// TwinCAT 3 PLC project Main
// ProgramVersion: 3.1.4024.0
// libraries:
//   Tc2_Standard, * (Beckhoff Automation GmbH)
//   Tc2_System, * (Beckhoff Automation GmbH)
//   Tc2_Utilities, * (Beckhoff Automation GmbH)
//   Tc3_Module, * (Beckhoff Automation GmbH)
//   TcUnit, * (www.tcunit.org)
//   mobject-core,0.5.0,mobject
//   mobject-graph-plc-pack,0.15.0,mobject
// project tree:
//   / PlcTask.TcTTO (not stored)
//   POUs/ MAIN.TcPOU
//   Tests/Alias/ _FLOAT_TestSuite.TcPOU (not stored), _HRESULT_TestSuite.TcPOU
//   Tests/Arrays/ _Array0to7OfByte_TestSuite.TcPOU
//   Tests/Enums/ _E_TcEventClass_TestSuite.TcPOU
//   Tests/Structs/ _GUID_TestSuite.TcPOU, _TIMESTRUCT_TestSuite.TcPOU
// real-time tasks:
//   TASK PlcTask: cycle T#10ms, priority 20, ADS port 350

// ---- POUs/MAIN.TcPOU
PROGRAM MAIN
VAR
	
	//alias
    _FLOAT_TestSuite : _FLOAT_TestSuite;
	_HRESULT_TestSuite : _HRESULT_TestSuite;
	
	// arrays
	_Array0to7OfByte_TestSuite : _Array0to7OfByte_TestSuite;
    
	// struct
	_TIMESTRUCT_TestSuite : _TIMESTRUCT_TestSuite;
	_GUID_TestSuite : _GUID_TestSuite;
	
	// enums
	_E_TcEventClass_TestSuite : _E_TcEventClass_TestSuite;
	
END_VAR

TcUnit.RUN();

END_PROGRAM

// ---- Tests/Alias/_HRESULT_TestSuite.TcPOU
FUNCTION_BLOCK _HRESULT_TestSuite EXTENDS TcUnit.FB_TestSuite
VAR
END_VAR

TestAddress();
TestClearReference();
TestClone();
TestTypeNameReturnsExpected();
TestIdentifierReturnsExpected();
TestMakeReferenceToFollowsReference();
TestMakeReferenceToUpdatesReference();
TestSize();
TestValueReturnsExpectedAfterInit();
TestValueReturnsExpectedAfterChange();
TestSerializeTypeWith();
TestSerializeWith();
TestTryDeserializeFrom();
TestTryMakeReferenceToFollowsReference();
TestTryMakeReferenceToUpdatesReference();

METHOD PUBLIC TestAddress
VAR
    _type : _HRESULT(S_OK);
    notExpected : PVOID := 0;
    actual : PVOID;
END_VAR
TEST('TestAddress');

actual := _type.Address;

AssertFalse(
    Condition := (notExpected = actual),
    Message := 'Type did not return a valid address.'
);

TEST_FINISHED();
END_METHOD

METHOD PUBLIC TestClearReference
VAR
    _type : _HRESULT(S_OK);
	target : HRESULT := S_OK;
    expected : HRESULT := S_OK;
    actual : HRESULT;
END_VAR
TEST('TestClearReference');

_type.MakeReferenceTo(target);
_type.ClearReference();
target := S_FALSE;

actual := _type.Value;

AssertEquals(
    Expected := expected,
    Actual := actual,
    Message := 'Value did not follow target change'
);

TEST_FINISHED();
END_METHOD

METHOD PUBLIC TestClone
VAR
    _type : _HRESULT(S_OK);
	clone : I_Datatype;
	isValidClone : BOOL;
	compareResult : DINT;
END_VAR
TEST('TestClone');

clone := _type.Clone();

isValidClone := clone <> 0;

IF isValidClone THEN
	compareResult := memcmp(_type.Address, clone.Address, clone.Size);
END_IF

AssertTrue(
	Condition := isValidClone,
	Message := 'Clone did not produce a clone'
);

AssertEquals_DINT(
	Expected := 0,
    Actual := compareResult,
    Message := 'Clone did not return a valid clone.'
);

clone.Dispose();

TEST_FINISHED();
END_METHOD

METHOD PUBLIC TestIdentifierReturnsExpected
VAR
    _type : _HRESULT(S_OK);
    expected : STRING := 'HRESULT';
    actual : STRING;
END_VAR
TEST('TestIdentifierReturnsExpected');

actual := _type.Identifier;

AssertEquals_STRING(
    Expected := expected,
    Actual := actual,
    Message := 'Type did not return correct iec type.'
);

TEST_FINISHED();
END_METHOD

METHOD PUBLIC TestMakeReferenceToFollowsReference
VAR
    _type : _HRESULT(S_OK);
	target : HRESULT := S_OK;
    expected : HRESULT := S_FALSE;
    actual : HRESULT;
END_VAR
TEST('TestMakeReferenceToFollowsReference');

_type.MakeReferenceTo(target);
target := S_FALSE;

actual := _type.Value;

AssertEquals(
    Expected := expected,
    Actual := actual,
    Message := 'Value did not follow target change'
);

TEST_FINISHED();
END_METHOD

METHOD PUBLIC TestMakeReferenceToUpdatesReference
VAR
    _type : _HRESULT(S_OK);
	target : HRESULT := S_OK;
    expected : HRESULT := S_FALSE;
    actual : HRESULT;
END_VAR
TEST('TestMakeReferenceToUpdatesReference');

_type.MakeReferenceTo(target);
_type.Value := S_FALSE;

actual := target;

AssertEquals(
    Expected := expected,
    Actual := actual,
    Message := 'Value did not update target'
);

TEST_FINISHED();
END_METHOD

METHOD PUBLIC TestSerializeTypeWith
VAR
    _type : _HRESULT(S_OK);
    serializer : JsonSerializer;
    expected : STRING(500) := '{"typeName":"ALIAS","identifier":"HRESULT","baseDatatype":{"typeName":"DINT","minValue":-2147483648,"maxValue":2147483647,"isSigned":true,"isFloat":false}}';
    actual : STRING(500);
END_VAR
TEST('TestSerializeTypeWith');

serializer.Reset();
_type.SerializeTypeWith(serializer);
serializer.TryGetSerializedData(ADR(actual), SIZEOF(actual));

AssertEquals_STRING(
    Expected := expected,
    Actual := actual,
    Message := 'Serialization of type did not return correct string.'
);

TEST_FINISHED();
END_METHOD

METHOD PUBLIC TestSerializeWith
VAR
    _type : _HRESULT(S_FALSE);
    serializer : JsonSerializer;
    expected : STRING := '1';
    actual : STRING(500);
END_VAR
TEST('TestSerializeWith');

serializer.Reset();
_type.SerializeWith(serializer);
serializer.TryGetSerializedData(ADR(actual), SIZEOF(actual));

AssertEquals_STRING(
    Expected := expected,
    Actual := actual,
    Message := 'Serialization of type data did not return correct string.'
);

TEST_FINISHED();
END_METHOD

METHOD PUBLIC TestSize
VAR
    _type : _HRESULT(S_OK);
    expected : UDINT := SIZEOF(HRESULT);
    actual : UDINT;
END_VAR
TEST('TestSize');

actual := _type.Size;

AssertEquals_UDINT(
    Expected := Expected,
    Actual := actual,
    Message := 'Type did not return the correct size.'
);

TEST_FINISHED();
END_METHOD

METHOD PUBLIC TestTryDeserializeFrom
VAR
    deserializer : JsonDeserializer;
    feedback : DeserializerFeedback;
    json : STRING := '0';
    _type : _HRESULT(S_OK);
    expected : HRESULT := S_OK;
    actual : HRESULT;
 END_VAR
TEST('TestTryDeserializeFrom');

deserializer.Reset();
deserializer.TryLoad(json);
_type.TryDeserializeFrom(Deserializer, Feedback);

actual := _type.Value;

AssertEquals(
    Expected := expected,
    Actual := actual,
    Message := 'Type did not deserialize correctly.'
);

TEST_FINISHED();
END_METHOD

METHOD PUBLIC TestTryMakeReferenceToFollowsReference
VAR
    _type : _HRESULT(S_OK);
	target : _HRESULT(S_OK);
    expected : HRESULT := S_FALSE;
    actual : HRESULT;
END_VAR
TEST('TestTryMakeReferenceToFollowsReference');

_type.TryMakeReferenceTo(target);
target.Value := S_FALSE;

actual := _type.Value;

AssertEquals(
    Expected := expected,
    Actual := actual,
    Message := 'Value did not follow target change'
);

TEST_FINISHED();
END_METHOD

METHOD PUBLIC TestTryMakeReferenceToUpdatesReference
VAR
    _type : _HRESULT(S_OK);
	target : _HRESULT(S_OK);
    expected : HRESULT := S_FALSE;
    actual : HRESULT;
END_VAR
TEST('TestTryMakeReferenceToUpdatesReference');

_type.TryMakeReferenceTo(target);
_type.Value := S_FALSE;

actual := target.Value;

AssertEquals(
    Expected := expected,
    Actual := actual,
    Message := 'Value did not update target'
);

TEST_FINISHED();
END_METHOD

METHOD PUBLIC TestTypeNameReturnsExpected
VAR
    _type : _HRESULT(S_OK);
    expected : STRING := 'ALIAS';
    actual : STRING;
END_VAR
TEST('TestTypeNameReturnsExpected');

actual := _type.TypeName;

AssertEquals_STRING(
    Expected := expected,
    Actual := actual,
    Message := 'Type did not return correct iec type.'
);

TEST_FINISHED();
END_METHOD

METHOD PUBLIC TestValueReturnsExpectedAfterChange
VAR
    _type : _HRESULT(S_OK);
    expected : HRESULT := S_FALSE;
    actual : HRESULT;
END_VAR
TEST('TestValueReturnsExpectedAfterChange');

_type.Value := S_FALSE;

actual := _type.Value;

AssertEquals(
    Expected := expected,
    Actual := actual,
    Message := 'Expected value not returned after change.'
);

TEST_FINISHED();
END_METHOD

METHOD PUBLIC TestValueReturnsExpectedAfterInit
VAR
    _type : _HRESULT(S_FALSE);
    expected : HRESULT := S_FALSE;
    actual : HRESULT;
END_VAR
TEST('TestValueReturnsExpectedAfterInit');

actual := _type.Value;

AssertEquals(
    Expected := expected,
    Actual := actual,
    Message := 'Expected value not returned after Init.'
);

TEST_FINISHED();
END_METHOD

END_FUNCTION_BLOCK

// ---- Tests/Arrays/_Array0to7OfByte_TestSuite.TcPOU
FUNCTION_BLOCK _Array0to7OfByte_TestSuite EXTENDS TcUnit.FB_TestSuite
VAR
END_VAR

TestAddress();
TestBaseDatatype();
TestClearReference();
TestClone();
TestTypeNameReturnsExpected();
TestIdentifierReturnsExpected();
TestLength();
TestLowerBound();
TestLowerBoundWithInvalidDimention();
TestMakeReferenceToFollowsReference();
TestMakeReferenceToUpdatesReference();
TestSize();
TestSerializeTypeWith();
TestSerializeWith();
TestTryDeserializeFrom();
TestTryGetElementAsDatatypeWithInvalidDimentionTooBig();
TestTryGetElementAsDatatypeWithInvalidDimentionTooSmall();
TestTryMakeReferenceToFollowsReference();
TestTryMakeReferenceToUpdatesReference();
TestUpperBound();
TestUpperBoundWithInvalidDimention();
TestValueReturnsExpectedAfterChange();

METHOD PUBLIC TestAddress
VAR
    _type : _Array0to7OfByte;
    notExpected : PVOID := 0;
    actual : PVOID;
END_VAR
TEST('TestAddress');

actual := _type.Address;

AssertFalse(
    Condition := (notExpected = actual),
    Message := 'Type did not return a valid address.'
);

TEST_FINISHED();
END_METHOD

METHOD PUBLIC TestBaseDatatype
VAR
    _type : _Array0to7OfByte;
    expected : T_MAXSTRING := 'BYTE';
    actual : T_MAXSTRING;
END_VAR
TEST('TestBaseDatatype');

actual := _type.BaseDatatype.TypeName;

AssertEquals_STRING(
    Expected := expected,
    Actual := actual,
    Message := 'Type did not return the correct base type'
);

TEST_FINISHED();
END_METHOD

METHOD PUBLIC TestClearReference
VAR
    _type : _Array0to7OfByte;
	target : ARRAY [0..7] OF BYTE;
    expected : ARRAY [0..7] OF BYTE := [0,0,0,0,0,0,0,0];
    actual : ARRAY [0..7] OF BYTE;
END_VAR
TEST('TestClearReference');

_type.MakeReferenceTo(target);
_type.ClearReference();
target[5] := 123;

actual := _type.Value;

AssertEquals(
    Expected := expected,
    Actual := actual,
    Message := 'Value incorrectly followed target change'
);

TEST_FINISHED();
END_METHOD

METHOD PUBLIC TestClone
VAR
    _type : _Array0to7OfByte;
	clone : I_Datatype;
	isValidClone : BOOL;
	compareResult : DINT;
END_VAR
TEST('TestClone');

clone := _type.Clone();

isValidClone := clone <> 0;

IF isValidClone THEN
	compareResult := memcmp(_type.Address, clone.Address, clone.Size);
END_IF

AssertTrue(
	Condition := isValidClone,
	Message := 'Clone did not produce a clone'
);

AssertEquals_DINT(
	Expected := 0,
    Actual := compareResult,
    Message := 'Clone did not return a valid clone.'
);

clone.Dispose();

TEST_FINISHED();
END_METHOD

METHOD PUBLIC TestIdentifierReturnsExpected
VAR
    _type : _Array0to7OfByte;
    expected : STRING := 'ARRAY [0..7] OF BYTE';
    actual : STRING;
END_VAR
TEST('TestIdentifierReturnsExpected');

actual := _type.Identifier;

AssertEquals_STRING(
    Expected := expected,
    Actual := actual,
    Message := 'Type did not return correct iec type.'
);

TEST_FINISHED();
END_METHOD

METHOD PUBLIC TestLength
VAR
    _type : _Array0to7OfByte;
    expected : UDINT := 8;
    actual : UDINT;
END_VAR
TEST('TestLength');

actual := _type.Length;

AssertEquals_UDINT(
    Expected := Expected,
    Actual := actual,
    Message := 'Type did not return the correct array length.'
);

TEST_FINISHED();
END_METHOD

METHOD PUBLIC TestLowerBound
VAR
    _type : _Array0to7OfByte;
    expected : DINT := 0;
    actual : DINT;
	ok : BOOL;
END_VAR
TEST('TestLowerBound');

ok := _type.TryGetLowerBound(1, actual);

AssertTrue(
    Condition := ok,
    Message := 'Type did not indicate that lower bound was possible to retreive.'
);

AssertEquals_DINT(
    Expected := Expected,
    Actual := actual,
    Message := 'Type did not return the correct array lower bound.'
);

TEST_FINISHED();
END_METHOD

METHOD PUBLIC TestLowerBoundWithInvalidDimention
VAR
    _type : _Array0to7OfByte;
    actual : DINT;
	result : BOOL;
END_VAR
TEST('TestLowerBoundWithInvalidDimention');

result := _type.TryGetLowerBound(2, actual);

AssertFalse(
    Condition := result,
    Message := 'Type did not indicate that the dimention was invalid'
);

TEST_FINISHED();
END_METHOD

METHOD PUBLIC TestMakeReferenceToFollowsReference
VAR
	_type : _Array0to7OfByte;
	target : ARRAY [0..7] OF BYTE;
    expected : ARRAY [0..7] OF BYTE := [1,2,3,4,5,6,7,8];
    actual : ARRAY [0..7] OF BYTE;
END_VAR
TEST('TestMakeReferenceToFollowsReference');

_type.MakeReferenceTo(target);
target[0] := 1;
target[1] := 2;
target[2] := 3;
target[3] := 4;
target[4] := 5;
target[5] := 6;
target[6] := 7;
target[7] := 8;

actual := _type.Value;

AssertEquals(
    Expected := expected,
    Actual := actual,
    Message := 'Value did not follow target change'
);

TEST_FINISHED();
END_METHOD

METHOD PUBLIC TestMakeReferenceToUpdatesReference
VAR
	_type : _Array0to7OfByte;
	target : ARRAY [0..7] OF BYTE;
    expected : ARRAY [0..7] OF BYTE := [1,2,3,4,5,6,7,8];
    actual : ARRAY [0..7] OF BYTE;
END_VAR
TEST('TestMakeReferenceToUpdatesReference');

_type.MakeReferenceTo(target);
target[0] := 1;
target[1] := 2;
target[2] := 3;
target[3] := 4;
target[4] := 5;
target[5] := 6;
target[6] := 7;
target[7] := 8;

actual := target;

AssertEquals(
    Expected := expected,
    Actual := actual,
    Message := 'Value did not update target'
);

TEST_FINISHED();
END_METHOD

METHOD PUBLIC TestSerializeTypeWith
VAR
    _type : _Array0to7OfByte;
    serializer : JsonSerializer;
    expected : STRING(1000) := '{"typeName":"ARRAY","identifier":"ARRAY [0..7] OF BYTE","baseType":{"typeName":"BYTE","minValue":0,"maxValue":255,"isSigned":false,"isFloat":false}}';
    actual : STRING(1000);
END_VAR
TEST('TestSerializeTypeWith');

serializer.Reset();
_type.SerializeTypeWith(serializer);
serializer.TryGetSerializedData(ADR(actual), SIZEOF(actual));

AssertEquals_STRING(
    Expected := expected,
    Actual := actual,
    Message := 'Serialization of type did not return correct string.'
);

TEST_FINISHED();
END_METHOD

METHOD PUBLIC TestSerializeWith
VAR
    _type : _Array0to7OfByte;
    serializer : JsonSerializer;
    expected : STRING(500) := '[1,2,3,4,5,6,7,8]';
    actual : STRING(500);
END_VAR
TEST('TestSerializeWith');

_type.Value[0] := 1;
_type.Value[1] := 2;
_type.Value[2] := 3;
_type.Value[3] := 4;
_type.Value[4] := 5;
_type.Value[5] := 6;
_type.Value[6] := 7;
_type.Value[7] := 8;

serializer.Reset();
_type.SerializeWith(serializer);
serializer.TryGetSerializedData(ADR(actual), SIZEOF(actual));

AssertEquals_STRING(
    Expected := expected,
    Actual := actual,
    Message := 'Serialization of type data did not return correct string.'
);

TEST_FINISHED();
END_METHOD

METHOD PUBLIC TestSize
VAR
    _type : _Array0to7OfByte;
	example : ARRAY [0..7] OF BYTE;
    expected : UDINT := SIZEOF(example);
    actual : UDINT;
END_VAR
TEST('TestSize');

actual := _type.Size;

AssertEquals_UDINT(
    Expected := Expected,
    Actual := actual,
    Message := 'Type did not return the correct size.'
);

TEST_FINISHED();
END_METHOD

METHOD PUBLIC TestTryDeserializeFrom
VAR
    deserializer : JsonDeserializer;
    feedback : DeserializerFeedback;
    json : STRING(500) := '[1,2,3,4,5,6,7,8]';
    _type : _Array0to7OfByte;
    expected :  ARRAY [0..7] OF BYTE := [1,2,3,4,5,6,7,8];
    actual : ARRAY [0..7] OF BYTE;
 END_VAR
TEST('TestTryDeserializeFrom');

deserializer.Reset();
deserializer.TryLoad(json);
_type.TryDeserializeFrom(Deserializer, Feedback);

actual := _type.Value;

AssertEquals(
    Expected := expected,
    Actual := actual,
    Message := 'Type did not deserialize correctly.'
);

TEST_FINISHED();
END_METHOD

METHOD PUBLIC TestTryGetElementAsDatatypeWithInvalidDimentionTooBig
VAR
    _type : _Array0to7OfByte;
    actual : I_Datatype;
	result : BOOL;
END_VAR
TEST('TestTryGetElementAsDatatypeWithInvalidDimentionTooBig');

result := _type.TryGetElementAsDatatypeByIndex(11, actual);

AssertFalse(
    Condition := result,
    Message := 'Type did not indicate that the dimention was invalid'
);

TEST_FINISHED();
END_METHOD

METHOD PUBLIC TestTryGetElementAsDatatypeWithInvalidDimentionTooSmall
VAR
    _type : _Array0to7OfByte;
    actual : I_Datatype;
	result : BOOL;
END_VAR
TEST('TestTryGetElementAsDatatypeWithInvalidDimentionTooSmall');

result := _type.TryGetElementAsDatatypeByIndex(-1, actual);

AssertFalse(
    Condition := result,
    Message := 'Type did not indicate that the dimention was invalid'
);

TEST_FINISHED();
END_METHOD

METHOD PUBLIC TestTryMakeReferenceToFollowsReference
VAR
    _type : _Array0to7OfByte;
	target : _Array0to7OfByte;
    expected : ARRAY [0..7] OF BYTE := [1,2,3,4,5,6,7,8];
    actual :  ARRAY [0..7] OF BYTE;
END_VAR
TEST('TestTryMakeReferenceToFollowsReference');

_type.TryMakeReferenceTo(target);
target.Value[0] := 1;
target.Value[1] := 2;
target.Value[2] := 3;
target.Value[3] := 4;
target.Value[4] := 5;
target.Value[5] := 6;
target.Value[6] := 7;
target.Value[7] := 8;

actual := _type.Value;

AssertEquals(
    Expected := expected,
    Actual := actual,
    Message := 'Value did not follow target change'
);

TEST_FINISHED();
END_METHOD

METHOD PUBLIC TestTryMakeReferenceToUpdatesReference
VAR
    _type : _Array0to7OfByte;
	target : _Array0to7OfByte;
    expected : ARRAY [0..7] OF BYTE := [1,2,3,4,5,6,7,8];
    actual :  ARRAY [0..7] OF BYTE;
END_VAR
TEST('TestTryMakeReferenceToUpdatesReference');

_type.TryMakeReferenceTo(target);
_type.Value[0] := 1;
_type.Value[1] := 2;
_type.Value[2] := 3;
_type.Value[3] := 4;
_type.Value[4] := 5;
_type.Value[5] := 6;
_type.Value[6] := 7;
_type.Value[7] := 8;

actual := target.Value;

AssertEquals(
    Expected := expected,
    Actual := actual,
    Message := 'Value did not update target'
);

TEST_FINISHED();
END_METHOD

METHOD PUBLIC TestTypeNameReturnsExpected
VAR
    _type : _Array0to7OfByte;
    expected : STRING := 'ARRAY';
    actual : STRING;
END_VAR
TEST('TestTypeNameReturnsExpected');

actual := _type.TypeName;

AssertEquals_STRING(
    Expected := expected,
    Actual := actual,
    Message := 'Type did not return correct iec type.'
);

TEST_FINISHED();
END_METHOD

METHOD PUBLIC TestUpperBound
VAR
    _type : _Array0to7OfByte;
    expected : DINT := 7;
    actual : DINT;
	ok : BOOL;
END_VAR
TEST('TestUpperBound');

ok := _type.TryGetUpperBound(1, actual);

AssertTrue(
    Condition := ok,
    Message := 'Type did not indicate that upper bound was possible to retreive.'
);

AssertEquals_DINT(
    Expected := Expected,
    Actual := actual,
    Message := 'Type did not return the correct array upper bound.'
);

TEST_FINISHED();
END_METHOD

METHOD PUBLIC TestUpperBoundWithInvalidDimention
VAR
    _type : _Array0to7OfByte;
    actual : DINT;
	result : BOOL;
END_VAR
TEST('TestUpperBoundWithInvalidDimention');

result := _type.TryGetUpperBound(2, actual);

AssertFalse(
    Condition := result,
    Message := 'Type did not indicate that the dimention was invalid'
);

TEST_FINISHED();
END_METHOD

METHOD PUBLIC TestValueReturnsExpectedAfterChange
VAR
    _type : _Array0to7OfByte;
	value : ARRAY [0..7] OF BYTE := [1,2,3,4,5,6,7,8];
    expected : ARRAY [0..7] OF BYTE := [1,2,3,4,5,6,7,8];
    actual :  ARRAY [0..7] OF BYTE;
END_VAR
TEST('TestValueReturnsExpectedAfterChange');

_type.Value := value;
actual := _type.Value;

AssertEquals(
    Expected := expected,
    Actual := actual,
    Message := 'Expected value not returned after change.'
);

TEST_FINISHED();
END_METHOD

END_FUNCTION_BLOCK

// ---- Tests/Structs/_TIMESTRUCT_TestSuite.TcPOU
FUNCTION_BLOCK _TIMESTRUCT_TestSuite EXTENDS TcUnit.FB_TestSuite
VAR
END_VAR

TestAddress();
TestClearReference();
TestClone();
TestTypeNameReturnsExpected();
TestIdentifierReturnsExpected();
TestMakeReferenceToFollowsReference();
TestMakeReferenceToUpdatesReference();
TestSize();
TestValueReturnsExpectedAfterChange();
TestSerializeTypeWith();
TestSerializeWith();
TestTryDeserializeFrom();
TestTryMakeReferenceToFollowsReference();
TestTryMakeReferenceToUpdatesReference();

METHOD PUBLIC TestAddress
VAR
    _type : _TIMESTRUCT;
    notExpected : PVOID := 0;
    actual : PVOID;
END_VAR
TEST('TestAddress');

actual := _type.Address;

AssertFalse(
    Condition := (notExpected = actual),
    Message := 'Type did not return a valid address.'
);

TEST_FINISHED();
END_METHOD

METHOD PUBLIC TestClearReference
VAR
    _type : _TIMESTRUCT;
	target : TIMESTRUCT;
    expected : TIMESTRUCT;
    actual : TIMESTRUCT;
END_VAR
TEST('TestClearReference');

_type.MakeReferenceTo(target);
_type.ClearReference();
target.wDay := 2;

actual := _type.Value;

AssertEquals(
    Expected := expected,
    Actual := actual,
    Message := 'Value did not follow target change'
);

TEST_FINISHED();
END_METHOD

METHOD PUBLIC TestClone
VAR
    _type : _TIMESTRUCT;
	clone : I_Datatype;
	isValidClone : BOOL;
	compareResult : DINT;
END_VAR
TEST('TestClone');

clone := _type.Clone();

isValidClone := clone <> 0;

IF isValidClone THEN
	compareResult := memcmp(_type.Address, clone.Address, clone.Size);
END_IF

AssertTrue(
	Condition := isValidClone,
	Message := 'Clone did not produce a clone'
);

AssertEquals_DINT(
	Expected := 0,
    Actual := compareResult,
    Message := 'Clone did not return a valid clone.'
);

clone.Dispose();

TEST_FINISHED();
END_METHOD

METHOD PUBLIC TestIdentifierReturnsExpected
VAR
    _type : _TIMESTRUCT;
    expected : STRING := 'TIMESTRUCT';
    actual : STRING;
END_VAR
TEST('TestIdentifierReturnsExpected');

actual := _type.Identifier;

AssertEquals_STRING(
    Expected := expected,
    Actual := actual,
    Message := 'Type did not return correct iec type.'
);

TEST_FINISHED();
END_METHOD

METHOD PUBLIC TestMakeReferenceToFollowsReference
VAR
    _type : _TIMESTRUCT;
	target : TIMESTRUCT;
    expected : TIMESTRUCT := (wDay := 2);
    actual : TIMESTRUCT;
END_VAR
TEST('TestMakeReferenceToFollowsReference');

_type.MakeReferenceTo(target);
target.wDay := 2;

actual := _type.Value;

AssertEquals(
    Expected := expected,
    Actual := actual,
    Message := 'Value did not follow target change'
);

TEST_FINISHED();
END_METHOD

METHOD PUBLIC TestMakeReferenceToUpdatesReference
VAR
    _type : _TIMESTRUCT;
	target : TIMESTRUCT;
    expected : TIMESTRUCT := (wDay := 2);
    actual : TIMESTRUCT;
END_VAR
TEST('TestMakeReferenceToUpdatesReference');

_type.MakeReferenceTo(target);
_type.wDay.Value := 2;

actual := target;

AssertEquals(
    Expected := expected,
    Actual := actual,
    Message := 'Value did not update target'
);

TEST_FINISHED();
END_METHOD

METHOD PUBLIC TestSerializeTypeWith
VAR
    _type : _TIMESTRUCT;
    serializer : JsonSerializer;
    expected : STRING(1000) := '{"typeName":"STRUCT","identifier":"TIMESTRUCT","members":{"wYear":{"typeName":"WORD","minValue":0,"maxValue":65535,"isSigned":false,"isFloat":false},"wMonth":{"typeName":"WORD","minValue":0,"maxValue":65535,"isSigned":false,"isFloat":false},"wDayOfWeek":{"typeName":"WORD","minValue":0,"maxValue":65535,"isSigned":false,"isFloat":false},"wDay":{"typeName":"WORD","minValue":0,"maxValue":65535,"isSigned":false,"isFloat":false},"wHour":{"typeName":"WORD","minValue":0,"maxValue":65535,"isSigned":false,"isFloat":false},"wMinute":{"typeName":"WORD","minValue":0,"maxValue":65535,"isSigned":false,"isFloat":false},"wSecond":{"typeName":"WORD","minValue":0,"maxValue":65535,"isSigned":false,"isFloat":false},"wMilliseconds":{"typeName":"WORD","minValue":0,"maxValue":65535,"isSigned":false,"isFloat":false}}}';
    actual : STRING(1000);
END_VAR
TEST('TestSerializeTypeWith');

serializer.Reset();
_type.SerializeTypeWith(serializer);
serializer.TryGetSerializedData(ADR(actual), SIZEOF(actual));

AssertEquals_STRING(
    Expected := expected,
    Actual := actual,
    Message := 'Serialization of type did not return correct string.'
);

TEST_FINISHED();
END_METHOD

METHOD PUBLIC TestSerializeWith
VAR
    _type : _TIMESTRUCT;
    serializer : JsonSerializer;
    expected : STRING(500) := '{"wYear":2000,"wMonth":1,"wDayOfWeek":2,"wDay":3,"wHour":4,"wMinute":5,"wSecond":6,"wMilliseconds":7}';
    actual : STRING(500);
END_VAR
TEST('TestSerializeWith');

_type.wYear.Value := 2000;
_type.wMonth.Value := 1;
_type.wDayOfWeek.Value := 2;
_type.wDay.Value := 3;
_type.wHour.Value := 4;
_type.wMinute.Value := 5;
_type.wSecond.Value := 6;
_type.wMilliseconds.Value := 7;

serializer.Reset();
_type.SerializeWith(serializer);
serializer.TryGetSerializedData(ADR(actual), SIZEOF(actual));

AssertEquals_STRING(
    Expected := expected,
    Actual := actual,
    Message := 'Serialization of type data did not return correct string.'
);

TEST_FINISHED();
END_METHOD

METHOD PUBLIC TestSize
VAR
    _type : _TIMESTRUCT;
    expected : UDINT := SIZEOF(TIMESTRUCT);
    actual : UDINT;
END_VAR
TEST('TestSize');

actual := _type.Size;

AssertEquals_UDINT(
    Expected := Expected,
    Actual := actual,
    Message := 'Type did not return the correct size.'
);

TEST_FINISHED();
END_METHOD

METHOD PUBLIC TestTryDeserializeFrom
VAR
    deserializer : JsonDeserializer;
    feedback : DeserializerFeedback;
    json : STRING(500) := '{"wDay":3,"wDayOfWeek":2,"wHour":4,"wMilliseconds":7,"wMinute":5,"wMonth":1,"wSecond":6,"wYear":2000}';
    _type : _TIMESTRUCT;
    expected : TIMESTRUCT := (wYear := 2000, wMonth := 1, wDayOfWeek := 2, wDay := 3, wHour := 4, wMinute := 5, wSecond := 6, wMilliseconds := 7);
    actual : TIMESTRUCT;
 END_VAR
TEST('TestTryDeserializeFrom');

deserializer.Reset();
deserializer.TryLoad(json);
_type.TryDeserializeFrom(Deserializer, Feedback);

actual := _type.Value;

AssertEquals(
    Expected := expected,
    Actual := actual,
    Message := 'Type did not deserialize correctly.'
);

TEST_FINISHED();
END_METHOD

METHOD PUBLIC TestTryMakeReferenceToFollowsReference
VAR
    _type : _TIMESTRUCT;
	target : _TIMESTRUCT;
    expected : TIMESTRUCT := (wDay := 2);
    actual : TIMESTRUCT;
END_VAR
TEST('TestTryMakeReferenceToFollowsReference');

_type.TryMakeReferenceTo(target);
target.wDay.Value := 2;

actual := _type.Value;

AssertEquals(
    Expected := expected,
    Actual := actual,
    Message := 'Value did not follow target change'
);

TEST_FINISHED();
END_METHOD

METHOD PUBLIC TestTryMakeReferenceToUpdatesReference
VAR
    _type : _TIMESTRUCT;
	target : _TIMESTRUCT;
    expected : TIMESTRUCT := (wDay := 2);
    actual : TIMESTRUCT;
END_VAR
TEST('TestTryMakeReferenceToUpdatesReference');

_type.TryMakeReferenceTo(target);
_type.wDay.Value := 2;

actual := target.Value;

AssertEquals(
    Expected := expected,
    Actual := actual,
    Message := 'Value did not update target'
);

TEST_FINISHED();
END_METHOD

METHOD PUBLIC TestTypeNameReturnsExpected
VAR
    _type : _TIMESTRUCT;
    expected : STRING := 'STRUCT';
    actual : STRING;
END_VAR
TEST('TestTypeNameReturnsExpected');

actual := _type.TypeName;

AssertEquals_STRING(
    Expected := expected,
    Actual := actual,
    Message := 'Type did not return correct iec type.'
);

TEST_FINISHED();
END_METHOD

METHOD PUBLIC TestValueReturnsExpectedAfterChange
VAR
    _type : _TIMESTRUCT;
	value : TIMESTRUCT := (wDay := 2);
    expected : TIMESTRUCT := (wDay := 2);
    actual : TIMESTRUCT;
END_VAR
TEST('TestValueReturnsExpectedAfterChange');

_type.Value := value;
actual := _type.Value;

AssertEquals(
    Expected := expected,
    Actual := actual,
    Message := 'Expected value not returned after change.'
);

TEST_FINISHED();
END_METHOD

END_FUNCTION_BLOCK

// ---- Tests/Structs/_GUID_TestSuite.TcPOU
FUNCTION_BLOCK _GUID_TestSuite EXTENDS TcUnit.FB_TestSuite
VAR
END_VAR

TestAddress();
TestClearReference();
TestClone();
TestTypeNameReturnsExpected();
TestIdentifierReturnsExpected();
TestMakeReferenceToFollowsReference();
TestMakeReferenceToUpdatesReference();
TestSize();
TestValueReturnsExpectedAfterChange();
TestSerializeTypeWith();
TestSerializeWith();
TestTryDeserializeFrom_String();
TestTryDeserializeFrom_Structure();
TestTryMakeReferenceToFollowsReference();
TestTryMakeReferenceToUpdatesReference();

METHOD PUBLIC TestAddress
VAR
    _type : _GUID;
    notExpected : PVOID := 0;
    actual : PVOID;
END_VAR
TEST('TestAddress');

actual := _type.Address;

AssertFalse(
    Condition := (notExpected = actual),
    Message := 'Type did not return a valid address.'
);

TEST_FINISHED();
END_METHOD

METHOD PUBLIC TestClearReference
VAR
    _type : _GUID;
	target : GUID;
    expected : GUID;
    actual : GUID;
END_VAR
TEST('TestClearReference');

_type.MakeReferenceTo(target);
_type.ClearReference();
target.Data1 := 123;

actual := _type.Value;

AssertEquals(
    Expected := expected,
    Actual := actual,
    Message := 'Value did not follow target change'
);

TEST_FINISHED();
END_METHOD

METHOD PUBLIC TestClone
VAR
    _type : _GUID;
	clone : I_Datatype;
	isValidClone : BOOL;
	compareResult : DINT;
END_VAR
TEST('TestClone');

clone := _type.Clone();

isValidClone := clone <> 0;

IF isValidClone THEN
	compareResult := memcmp(_type.Address, clone.Address, clone.Size);
END_IF

AssertTrue(
	Condition := isValidClone,
	Message := 'Clone did not produce a clone'
);

AssertEquals_DINT(
	Expected := 0,
    Actual := compareResult,
    Message := 'Clone did not return a valid clone.'
);

clone.Dispose();

TEST_FINISHED();
END_METHOD

METHOD PUBLIC TestIdentifierReturnsExpected
VAR
    _type : _GUID;
    expected : STRING := 'GUID';
    actual : STRING;
END_VAR
TEST('TestIdentifierReturnsExpected');

actual := _type.Identifier;

AssertEquals_STRING(
    Expected := expected,
    Actual := actual,
    Message := 'Type did not return correct iec type.'
);

TEST_FINISHED();
END_METHOD

METHOD PUBLIC TestMakeReferenceToFollowsReference
VAR
    _type : _GUID;
	target : GUID;
    expected : GUID := (Data1 := 1, Data2 := 2, Data3 := 3, Data4 := [4,5,6,7,8,9,10,11]);
    actual : GUID;
END_VAR
TEST('TestMakeReferenceToFollowsReference');

_type.MakeReferenceTo(target);
target.Data1 := 1;
target.Data2 := 2;
target.Data3 := 3;
target.Data4[0] := 4;
target.Data4[1] := 5;
target.Data4[2] := 6;
target.Data4[3] := 7;
target.Data4[4] := 8;
target.Data4[5] := 9;
target.Data4[6] := 10;
target.Data4[7] := 11;

actual := _type.Value;

AssertEquals(
    Expected := expected,
    Actual := actual,
    Message := 'Value did not follow target change'
);

TEST_FINISHED();
END_METHOD

METHOD PUBLIC TestMakeReferenceToUpdatesReference
VAR
    _type : _GUID;
	target : GUID;
    expected : GUID := (Data1 := 1, Data2 := 2, Data3 := 3, Data4 := [4,5,6,7,8,9,10,11]);
    actual : GUID;
END_VAR
TEST('TestMakeReferenceToUpdatesReference');

_type.MakeReferenceTo(target);
_type.Data1.Value := 1;
_type.Data2.Value := 2;
_type.Data3.Value := 3;
_type.Data4.Value[0] := 4;
_type.Data4.Value[1] := 5;
_type.Data4.Value[2] := 6;
_type.Data4.Value[3] := 7;
_type.Data4.Value[4] := 8;
_type.Data4.Value[5] := 9;
_type.Data4.Value[6] := 10;
_type.Data4.Value[7] := 11;

actual := target;

AssertEquals(
    Expected := expected,
    Actual := actual,
    Message := 'Value did not update target'
);

TEST_FINISHED();
END_METHOD

METHOD PUBLIC TestSerializeTypeWith
VAR
    _type : _GUID;
    serializer : JsonSerializer;
    expected : STRING(1000) := '{"typeName":"STRUCT","identifier":"GUID","members":{"Data1":{"typeName":"DWORD","minValue":0,"maxValue":4294967295,"isSigned":false,"isFloat":false},"Data2":{"typeName":"WORD","minValue":0,"maxValue":65535,"isSigned":false,"isFloat":false},"Data3":{"typeName":"WORD","minValue":0,"maxValue":65535,"isSigned":false,"isFloat":false},"Data4":{"typeName":"ARRAY","identifier":"ARRAY [0..7] OF BYTE","baseType":{"typeName":"BYTE","minValue":0,"maxValue":255,"isSigned":false,"isFloat":false}}}}';
    actual : STRING(1000);
END_VAR
TEST('TestSerializeTypeWith');

serializer.Reset();
_type.SerializeTypeWith(serializer);
serializer.TryGetSerializedData(ADR(actual), SIZEOF(actual));

AssertEquals_STRING(
    Expected := expected,
    Actual := actual,
    Message := 'Serialization of type did not return correct string.'
);

TEST_FINISHED();
END_METHOD

METHOD PUBLIC TestSerializeWith
VAR
    _type : _GUID;
    serializer : JsonSerializer;
    expected : STRING(500) := '{"Data1":1,"Data2":2,"Data3":3,"Data4":[4,5,6,7,8,9,10,11]}';
    actual : STRING(500);
END_VAR
TEST('TestSerializeWith');

_type.Data1.Value := 1;
_type.Data2.Value := 2;
_type.Data3.Value := 3;
_type.Data4.Value[0] := 4;
_type.Data4.Value[1] := 5;
_type.Data4.Value[2] := 6;
_type.Data4.Value[3] := 7;
_type.Data4.Value[4] := 8;
_type.Data4.Value[5] := 9;
_type.Data4.Value[6] := 10;
_type.Data4.Value[7] := 11;

serializer.Reset();
_type.SerializeWith(serializer);
serializer.TryGetSerializedData(ADR(actual), SIZEOF(actual));

AssertEquals_STRING(
    Expected := expected,
    Actual := actual,
    Message := 'Serialization of type data did not return correct string.'
);

TEST_FINISHED();
END_METHOD

METHOD PUBLIC TestSize
VAR
    _type : _GUID;
    expected : UDINT := SIZEOF(GUID);
    actual : UDINT;
END_VAR
TEST('TestSize');

actual := _type.Size;

AssertEquals_UDINT(
    Expected := Expected,
    Actual := actual,
    Message := 'Type did not return the correct size.'
);

TEST_FINISHED();
END_METHOD

METHOD PUBLIC TestTryDeserializeFrom_String
VAR
    deserializer : JsonDeserializer;
    feedback : DeserializerFeedback;
    json : STRING(500) := '"123e4567-e89b-12d3-a456-426655440000"';
    _type : _GUID;
    expected : GUID := (Data1:=16#123E4567, Data2:=16#E89B, Data3:=16#12D3, Data4:=[16#A4, 16#56, 16#42, 16#66, 16#55, 16#44, 16#00, 16#00]);
    actual : GUID;
 END_VAR
TEST('TestTryDeserializeFrom_String');

deserializer.Reset();
deserializer.TryLoad(json);
_type.TryDeserializeFrom(Deserializer, Feedback);

actual := _type.Value;

AssertEquals(
    Expected := expected,
    Actual := actual,
    Message := 'Type did not deserialize correctly.'
);

TEST_FINISHED();
END_METHOD

METHOD PUBLIC TestTryDeserializeFrom_Structure
VAR
    deserializer : JsonDeserializer;
    feedback : DeserializerFeedback;
    json : STRING(500) := '{"Data1":1,"Data2":2,"Data3":3,"Data4":[4,5,6,7,8,9,10,11]}';
    _type : _GUID;
    expected : GUID := (Data1 := 1, Data2 := 2, Data3 := 3, Data4 := [4,5,6,7,8,9,10,11]);
    actual : GUID;
 END_VAR
TEST('TestTryDeserializeFrom_Structure');

deserializer.Reset();
deserializer.TryLoad(json);
_type.TryDeserializeFrom(Deserializer, Feedback);

actual := _type.Value;

AssertEquals(
    Expected := expected,
    Actual := actual,
    Message := 'Type did not deserialize correctly.'
);

TEST_FINISHED();
END_METHOD

METHOD PUBLIC TestTryMakeReferenceToFollowsReference
VAR
    _type : _GUID;
	target : _GUID;
    expected : GUID := (Data1 := 1, Data2 := 2, Data3 := 3, Data4 := [4,5,6,7,8,9,10,11]);
    actual : GUID;
END_VAR
TEST('TestTryMakeReferenceToFollowsReference');

_type.TryMakeReferenceTo(target);
target.Data1.Value := 1;
target.Data2.Value := 2;
target.Data3.Value := 3;
target.Data4.Value[0] := 4;
target.Data4.Value[1] := 5;
target.Data4.Value[2] := 6;
target.Data4.Value[3] := 7;
target.Data4.Value[4] := 8;
target.Data4.Value[5] := 9;
target.Data4.Value[6] := 10;
target.Data4.Value[7] := 11;

actual := _type.Value;

AssertEquals(
    Expected := expected,
    Actual := actual,
    Message := 'Value did not follow target change'
);

TEST_FINISHED();
END_METHOD

METHOD PUBLIC TestTryMakeReferenceToUpdatesReference
VAR
    _type : _GUID;
	target : _GUID;
    expected : GUID := (Data1 := 1, Data2 := 2, Data3 := 3, Data4 := [4,5,6,7,8,9,10,11]);
    actual : GUID;
END_VAR
TEST('TestTryMakeReferenceToUpdatesReference');

_type.TryMakeReferenceTo(target);
_type.Data1.Value := 1;
_type.Data2.Value := 2;
_type.Data3.Value := 3;
_type.Data4.Value[0] := 4;
_type.Data4.Value[1] := 5;
_type.Data4.Value[2] := 6;
_type.Data4.Value[3] := 7;
_type.Data4.Value[4] := 8;
_type.Data4.Value[5] := 9;
_type.Data4.Value[6] := 10;
_type.Data4.Value[7] := 11;

actual := target.Value;

AssertEquals(
    Expected := expected,
    Actual := actual,
    Message := 'Value did not update target'
);

TEST_FINISHED();
END_METHOD

METHOD PUBLIC TestTypeNameReturnsExpected
VAR
    _type : _GUID;
    expected : STRING := 'STRUCT';
    actual : STRING;
END_VAR
TEST('TestTypeNameReturnsExpected');

actual := _type.TypeName;

AssertEquals_STRING(
    Expected := expected,
    Actual := actual,
    Message := 'Type did not return correct iec type.'
);

TEST_FINISHED();
END_METHOD

METHOD PUBLIC TestValueReturnsExpectedAfterChange
VAR
    _type : _GUID;
	value : GUID := (Data1 := 1, Data2 := 2, Data3 := 3, Data4 := [4,5,6,7,8,9,10,11]);
    expected : GUID := (Data1 := 1, Data2 := 2, Data3 := 3, Data4 := [4,5,6,7,8,9,10,11]);
    actual : GUID;
END_VAR
TEST('TestValueReturnsExpectedAfterChange');

_type.Value := value;
actual := _type.Value;

AssertEquals(
    Expected := expected,
    Actual := actual,
    Message := 'Expected value not returned after change.'
);

TEST_FINISHED();
END_METHOD

END_FUNCTION_BLOCK

// ---- Tests/Enums/_E_TcEventClass_TestSuite.TcPOU
FUNCTION_BLOCK _E_TcEventClass_TestSuite EXTENDS TcUnit.FB_TestSuite
VAR
END_VAR

TestAddress();
TestClearReference();
TestClone();
TestTypeNameReturnsExpected();
TestIdentifierReturnsExpected();
TestMakeReferenceToFollowsReference();
TestMakeReferenceToUpdatesReference();
TestSize();
TestValueReturnsExpectedAfterInit();
TestValueReturnsExpectedAfterChange();
TestSerializeTypeWith();
TestSerializeWith();
TestTryDeserializeFrom();
TestTryMakeReferenceToFollowsReference();
TestTryMakeReferenceToUpdatesReference();

METHOD PUBLIC TestAddress
VAR
    _type : _E_TcEventClass(E_TcEventClass.TCEVENTCLASS_NONE);
    notExpected : PVOID := 0;
    actual : PVOID;
END_VAR
TEST('TestAddress');

actual := _type.Address;

AssertFalse(
    Condition := (notExpected = actual),
    Message := 'Type did not return a valid address.'
);

TEST_FINISHED();
END_METHOD

METHOD PUBLIC TestClearReference
VAR
    _type : _E_TcEventClass(E_TcEventClass.TCEVENTCLASS_NONE);
	target : E_TcEventClass := E_TcEventClass.TCEVENTCLASS_NONE;
    expected : E_TcEventClass := E_TcEventClass.TCEVENTCLASS_NONE;
    actual : E_TcEventClass;
END_VAR
TEST('TestClearReference');

_type.MakeReferenceTo(target);
_type.ClearReference();
target := E_TcEventClass.TCEVENTCLASS_ALARM;

actual := _type.Value;

AssertEquals(
    Expected := expected,
    Actual := actual,
    Message := 'Value did not follow target change'
);

TEST_FINISHED();
END_METHOD

METHOD PUBLIC TestClone
VAR
    _type : _E_TcEventClass(E_TcEventClass.TCEVENTCLASS_NONE);
	clone : I_Datatype;
	isValidClone : BOOL;
	compareResult : DINT;
END_VAR
TEST('TestClone');

clone := _type.Clone();

isValidClone := clone <> 0;

IF isValidClone THEN
	compareResult := memcmp(_type.Address, clone.Address, clone.Size);
END_IF

AssertTrue(
	Condition := isValidClone,
	Message := 'Clone did not produce a clone'
);

AssertEquals_DINT(
	Expected := 0,
    Actual := compareResult,
    Message := 'Clone did not return a valid clone.'
);

clone.Dispose();

TEST_FINISHED();
END_METHOD

METHOD PUBLIC TestIdentifierReturnsExpected
VAR
    _type : _E_TcEventClass(E_TcEventClass.TCEVENTCLASS_NONE);;
    expected : STRING := 'E_TcEventClass';
    actual : STRING;
END_VAR
TEST('TestIdentifierReturnsExpected');

actual := _type.Identifier;

AssertEquals_STRING(
    Expected := expected,
    Actual := actual,
    Message := 'Type did not return correct iec type.'
);

TEST_FINISHED();
END_METHOD

METHOD PUBLIC TestMakeReferenceToFollowsReference
VAR
    _type : _E_TcEventClass(E_TcEventClass.TCEVENTCLASS_NONE);;
	target : E_TcEventClass := E_TcEventClass.TCEVENTCLASS_NONE;
    expected : E_TcEventClass := E_TcEventClass.TCEVENTCLASS_ALARM;
    actual : E_TcEventClass;
END_VAR
TEST('TestMakeReferenceToFollowsReference');

_type.MakeReferenceTo(target);
target := E_TcEventClass.TCEVENTCLASS_ALARM;

actual := _type.Value;

AssertEquals(
    Expected := expected,
    Actual := actual,
    Message := 'Value did not follow target change'
);

TEST_FINISHED();
END_METHOD

METHOD PUBLIC TestMakeReferenceToUpdatesReference
VAR
    _type : _E_TcEventClass(E_TcEventClass.TCEVENTCLASS_NONE);;
	target : E_TcEventClass := E_TcEventClass.TCEVENTCLASS_NONE;
    expected : E_TcEventClass := E_TcEventClass.TCEVENTCLASS_ALARM;
    actual : E_TcEventClass;
END_VAR
TEST('TestMakeReferenceToUpdatesReference');

_type.MakeReferenceTo(target);
_type.Value := E_TcEventClass.TCEVENTCLASS_ALARM;

actual := target;

AssertEquals(
    Expected := expected,
    Actual := actual,
    Message := 'Value did not update target'
);

TEST_FINISHED();
END_METHOD

METHOD PUBLIC TestSerializeTypeWith
VAR
    _type : _E_TcEventClass(E_TcEventClass.TCEVENTCLASS_NONE);
    serializer : JsonSerializer;
    expected : STRING(500) := '{"typeName":"ENUM","identifier":"E_TcEventClass","enumerations":["TCEVENTCLASS_NONE","TCEVENTCLASS_MAINTENANCE","TCEVENTCLASS_MESSAGE","TCEVENTCLASS_HINT","TCEVENTCLASS_STATEINFO","TCEVENTCLASS_INSTRUCTION","TCEVENTCLASS_WARNING","TCEVENTCLASS_ALARM","TCEVENTCLASS_PARAMERROR"],"baseType":{"typeName":"UINT","minValue":0,"maxValue":65535,"isSigned":false,"isFloat":false}}';
    actual : STRING(500);
END_VAR
TEST('TestSerializeTypeWith');

serializer.Reset();
_type.SerializeTypeWith(serializer);
serializer.TryGetSerializedData(ADR(actual), SIZEOF(actual));

AssertEquals_STRING(
    Expected := expected,
    Actual := actual,
    Message := 'Serialization of type did not return correct string.'
);

TEST_FINISHED();
END_METHOD

METHOD PUBLIC TestSerializeWith
VAR
    _type : _E_TcEventClass(E_TcEventClass.TCEVENTCLASS_ALARM);
    serializer : JsonSerializer;
    expected : STRING := '"TCEVENTCLASS_ALARM"';
    actual : STRING(500);
END_VAR
TEST('TestSerializeWith');

serializer.Reset();
_type.SerializeWith(serializer);
serializer.TryGetSerializedData(ADR(actual), SIZEOF(actual));

AssertEquals_STRING(
    Expected := expected,
    Actual := actual,
    Message := 'Serialization of type data did not return correct string.'
);

TEST_FINISHED();
END_METHOD

METHOD PUBLIC TestSize
VAR
    _type : _E_TcEventClass(E_TcEventClass.TCEVENTCLASS_NONE);;
    expected : UDINT := SIZEOF(E_TcEventClass);
    actual : UDINT;
END_VAR
TEST('TestSize');

actual := _type.Size;

AssertEquals_UDINT(
    Expected := Expected,
    Actual := actual,
    Message := 'Type did not return the correct size.'
);

TEST_FINISHED();
END_METHOD

METHOD PUBLIC TestTryDeserializeFrom
VAR
    deserializer : JsonDeserializer;
    feedback : DeserializerFeedback;
    json : STRING := '"TCEVENTCLASS_ALARM"';
    _type : _E_TcEventClass(E_TcEventClass.TCEVENTCLASS_NONE);
    expected : E_TcEventClass := E_TcEventClass.TCEVENTCLASS_ALARM;
    actual : E_TcEventClass;
 END_VAR
TEST('TestTryDeserializeFrom');

deserializer.Reset();
deserializer.TryLoad(json);
_type.TryDeserializeFrom(Deserializer, Feedback);

actual := _type.Value;

AssertEquals_LREAL(
    Expected := expected,
    Actual := actual,
    Delta := LREAL#0.001,
    Message := 'Type did not deserialize correctly.'
);

TEST_FINISHED();
END_METHOD

METHOD PUBLIC TestTryMakeReferenceToFollowsReference
VAR
    _type : _E_TcEventClass(E_TcEventClass.TCEVENTCLASS_NONE);;
	target : _E_TcEventClass(E_TcEventClass.TCEVENTCLASS_NONE);;
    expected : E_TcEventClass := E_TcEventClass.TCEVENTCLASS_ALARM;
    actual : E_TcEventClass;
END_VAR
TEST('TestTryMakeReferenceToFollowsReference');

_type.TryMakeReferenceTo(target);
target.Value := E_TcEventClass.TCEVENTCLASS_ALARM;

actual := _type.Value;

AssertEquals(
    Expected := expected,
    Actual := actual,
    Message := 'Value did not follow target change'
);

TEST_FINISHED();
END_METHOD

METHOD PUBLIC TestTryMakeReferenceToUpdatesReference
VAR
    _type : _E_TcEventClass(E_TcEventClass.TCEVENTCLASS_NONE);;
	target : _E_TcEventClass(E_TcEventClass.TCEVENTCLASS_NONE);;
    expected : E_TcEventClass := E_TcEventClass.TCEVENTCLASS_ALARM;
    actual : E_TcEventClass;
END_VAR
TEST('TestTryMakeReferenceToUpdatesReference');

_type.TryMakeReferenceTo(target);
_type.Value := E_TcEventClass.TCEVENTCLASS_ALARM;

actual := target.Value;

AssertEquals(
    Expected := expected,
    Actual := actual,
    Message := 'Value did not update target'
);

TEST_FINISHED();
END_METHOD

METHOD PUBLIC TestTypeNameReturnsExpected
VAR
    _type : _E_TcEventClass(E_TcEventClass.TCEVENTCLASS_NONE);;
    expected : STRING := 'ENUM';
    actual : STRING;
END_VAR
TEST('TestTypeNameReturnsExpected');

actual := _type.TypeName;

AssertEquals_STRING(
    Expected := expected,
    Actual := actual,
    Message := 'Type did not return correct iec type.'
);

TEST_FINISHED();
END_METHOD

METHOD PUBLIC TestValueReturnsExpectedAfterChange
VAR
    _type : _E_TcEventClass(E_TcEventClass.TCEVENTCLASS_NONE);;
    expected : E_TcEventClass := E_TcEventClass.TCEVENTCLASS_ALARM;
    actual : E_TcEventClass;
END_VAR
TEST('TestValueReturnsExpectedAfterChange');

_type.Value := E_TcEventClass.TCEVENTCLASS_ALARM;

actual := _type.Value;

AssertEquals(
    Expected := expected,
    Actual := actual,
    Message := 'Expected value not returned after change.'
);

TEST_FINISHED();
END_METHOD

METHOD PUBLIC TestValueReturnsExpectedAfterInit
VAR
    _type : _E_TcEventClass(E_TcEventClass.TCEVENTCLASS_ALARM);
    expected : E_TcEventClass := E_TcEventClass.TCEVENTCLASS_ALARM;
    actual : E_TcEventClass;
END_VAR
TEST('TestValueReturnsExpectedAfterInit');

actual := _type.Value;

AssertEquals(
    Expected := expected,
    Actual := actual,
    Message := 'Expected value not returned after Init.'
);

TEST_FINISHED();
END_METHOD

END_FUNCTION_BLOCK
